  rq_init_comm_if_connected(9, "1")
  rq_init_comm_if_connected(2, "2")
  rq_init_comm_if_connected(3, "3")
  rq_init_comm_if_connected(4, "4")
  rq_print_connected_grippers()
  rq_gripper_communication_thread = run rq_gripper_communication()
  set_closed_norm(100.0, 1)
  set_open_norm(0.0, 1)
  set_closed_mm(0.0, 1)
  set_open_mm(50.0, 1)
  set_closed_norm(100.0, 2)
  set_open_norm(0.0, 2)
  set_closed_mm(0.0, 2)
  set_open_mm(50.0, 2)
  set_closed_norm(100.0, 3)
  set_open_norm(0.0, 3)
  set_closed_mm(0.0, 3)
  set_open_mm(50.0, 3)
  set_closed_norm(100.0, 4)
  set_open_norm(0.0, 4)
  set_closed_mm(0.0, 4)
  set_open_mm(50.0, 4)
  rq_current_limit_enabled = False
  while(not rq_gripper_communication_thread_started):
      sleep(0.008)
  end
  # end: URCap Installation Node
  step_count_6f5ccb1a_e640_4da3_bfd2_40e239d724c0 = 0.0
  thread Step_Counter_Thread_dce1a192_0697_4136_975c_3f443e1826c0():
    while (True):
      step_count_6f5ccb1a_e640_4da3_bfd2_40e239d724c0 = step_count_6f5ccb1a_e640_4da3_bfd2_40e239d724c0 + 1.0
      sync()
    end
  end
  run Step_Counter_Thread_dce1a192_0697_4136_975c_3f443e1826c0()
  global Pallet_1_cnt1=1
  global Pallet_1_lct=1
  global Pallet_1_lno=1
  global Pallet_1_sep= False
  global Pallet_1_tct=1
  global ready_bottle_01_p=p[.390695686427, .546143722526, .354784252936, -1.202154726952, -2.902476248553, -.000065055908]
  global ready_bottle_01_q=[1.2121562957763672, -1.5242460531047364, -1.8409428596496582, -1.3471840184978028, 1.569084882736206, -2.714905563985006]
  global Approach_p=p[.547491153120, .654222384983, -.068387800069, 1.202193147572, 2.902469227050, .000121933136]
  global Approach_q=[1.079941749572754, -2.4608241520323695, -1.818922519683838, -0.4325900834849854, 1.569946050643921, -2.84857422510256]
  global ToolActionPoint_p=p[.547456310296, .654165465094, -.466875056309, 1.202132749463, 2.902463524491, -.000036040777]
  global ToolActionPoint_q=[1.0798958534460201, -3.092485844440475, -1.4373697255328164, -0.182578185020553, 1.5701887189532613, -2.8485011726798497]
  global Exit_1_p=p[.547471692821, .654225285966, -.113240204994, 1.202149918204, 2.902456390812, .000132406260]
  global Exit_1_q=[1.0799791934124974, -2.5300233635810003, -1.7983936890644978, -0.38391026593322053, 1.5699977418301563, -2.8485885945959932]
  global other_side_botl_p=p[-.131302644250, .581179310947, .471637250643, 1.202107245272, 2.902505419242, .000006210820]
  global other_side_botl_q=[2.0894155502319336, -1.3711059850505372, -1.7675957679748535, -1.573710104028219, 1.5691683292388916, -1.8372095266925257]
  global bottle_insert_p=p[-.131260964550, .980471403249, .471604896898, 1.202196404184, 2.902428691936, .000004532766]
  global bottle_insert_q=[1.880312442779541, -2.055948873559469, -0.9804320335388184, -1.6760550938048304, 1.5698020458221436, -2.045520607625143]
  global bottle_placed_p=p[-.131258911804, .980469640209, .306164973509, -1.202200405733, -2.902392835778, -.000046866587]
  global bottle_placed_q=[1.880561113357544, -2.0672136745848597, -1.2540980577468872, -1.3910349768451233, 1.5695239305496216, -2.0459168593036097]
  global bottle_left_p=p[-.131220480029, .980475238550, .407942093095, -1.202222478666, -2.902455166129, -.000055421236]
  global bottle_left_q=[1.8803844451904297, -2.050185819665426, -1.1006345748901367, -1.5615647596171875, 1.5696470737457275, -2.0457008520709437]
  global Waypoint_1_p=p[-.642107095425, .666282486477, .300000000000, .017110052262, 3.141514691896, -.000101435305]
  global Waypoint_1_q=[2.5268598030394767, -1.9627318786897927, -1.4187371386550547, -1.331007934561983, 1.5694235174349547, -2.174366234433882]
  global towards_tool_p=p[-.319103721707, .922274672984, .289488424593, -2.161715004584, 2.087946977393, .189764243643]
  global towards_tool_q=[2.109555244445801, -2.0061499081053675, -1.4868388175964355, -1.0633927148631592, 1.4768521785736084, 2.067403554916382]
  global opener_release_p=p[-.319041217029, .960983395363, .063631881470, -2.151377132576, 2.078331762283, .208011082729]
  global opener_release_q=[2.0912246704101562, -2.235462804833883, -1.5705714225769043, -0.7327280801585694, 1.4711558818817139, 2.0473134517669678]
  global Waypoint_2_p=p[-.130580669380, .976983076115, .465670208769, -1.211351089344, 1.169811544850, 1.192461372640]
  global Waypoint_2_q=[2.048638343811035, -1.9488769970335902, -1.9945645332336426, 0.8238295751759033, 1.0946009159088135, -4.7583046595202845]
  global Waypoint_3_p=p[-.130500299950, .978149746807, .289697846114, -1.201141215498, 1.186848407184, 1.212169596068]
  global Waypoint_3_q=[2.046792984008789, -2.209787984887594, -2.0315918922424316, 1.1217116552540283, 1.098623514175415, -4.7331653277026575]
  global Waypoint_4_p=p[-.128825153461, .982323687907, .290256016280, -.673557451662, .725956132353, 1.488202477063]
  global Waypoint_4_q=[1.9992650747299194, -2.605262895623678, -1.638580322265625, 1.8312062460133056, 1.2280412912368774, -4.949915353451864]
  global Waypoint_7_p=p[-.128786997274, .992110967731, .291362608216, -.774623003114, .830703590919, 1.448526193777]
  global Waypoint_7_q=[2.0093674659729004, -2.5409466228880824, -1.719653606414795, 1.7121011453815917, 1.185677170753479, -4.909483496342794]
  global Waypoint_5_p=p[-.130885594544, .990636414244, .290303660438, -1.093247620272, 1.014798422788, 1.277726987509]
  global Waypoint_5_q=[2.0226666927337646, -2.338917394677633, -1.9369897842407227, 1.357553406352661, 1.154337763786316, -4.854938570653097]
  global Waypoint_6_p=p[-.129580234191, .994111291374, .289563055839, -1.211278069791, 1.169892183217, 1.192387357827]
  global Waypoint_6_q=[2.0349059104919434, -2.223354002038473, -1.9993042945861816, 1.1026395994373779, 1.1086199283599854, -4.757455412541525]
  global put_opener_back_p=p[-.319099897221, .974896383339, .066796819335, -2.237817946884, 2.161546728532, .045382917786]
  global put_opener_back_q=[2.062997817993164, -2.282285829583639, -1.4317312240600586, -0.9614525598338624, 1.549813985824585, 2.027625799179077]
  global release_opener_p=p[-.319054355550, .963210691229, .061049693193, -2.161547074700, 2.088102897465, .189944602177]
  global release_opener_q=[2.0875582695007324, -2.2436233959593714, -1.555147647857666, -0.7554741662791749, 1.4804890155792236, 2.045177698135376]
  $ 2 "BeforeStart"
  $ 3 "ready_to_take≔ False "
  global ready_to_take=  False
  $ 4 "Loop_1≔0"
  global Loop_1=0
  $ 5 "Set"
  set_tcp(p[0.0,0.0,0.195,0.0,0.0,0.0])
  thread EventThread():
    while (True):
      if (ready_to_take ==   True  ):
        $ 316 "Set Start=On"
        set_standard_digital_out(0, True)
        $ 317 "Wait: 0.25"
        sleep(0.25)
        $ 318 "Set Start=Off"
        set_standard_digital_out(0, False)
        $ 319 "Wait: 0.25"
        sleep(0.25)
        $ 320 "If bottle_sensor≟ False "
        if (get_standard_digital_in(1) ==   False  ):
          $ 321 "ready_to_take≔ False "
          global ready_to_take=  False
        end
      end
      sync()
    end
  end
  eventThread = run EventThread()
  $ 6 "Robot Program"
  # begin: URCap Program Node
  #   Source: triplea-wingman, 1.4.0, tripleA robotics ApS
  #   Type: AAA - Tools
  $ 7 "AAA - Tools"
  # end: URCap Program Node
  # begin: URCap Program Node
  #   Source: triplea-wingman, 1.4.0, tripleA robotics ApS
  #   Type: AAA - Get Tool
  $ 28 "AAA - Get T2           "
  $ 29 "Waypoints" "noBreak"
  $ 30 "tool_id_3≔'4a342d3e-ee93-4452-a102-fbcfc7771081'" "noBreak"
  global tool_id_3="4a342d3e-ee93-4452-a102-fbcfc7771081"
  $ 31 "tool_w1_3≔aaa_get_w(1, tool_id_3)" "noBreak"
  global tool_w1_3= aaa_get_w (1, tool_id_3)
  $ 32 "tool_w2_3≔aaa_get_w(2, tool_id_3)" "noBreak"
  global tool_w2_3= aaa_get_w (2, tool_id_3)
  $ 33 "tool_w3_3≔aaa_get_w(3, tool_id_3)" "noBreak"
  global tool_w3_3= aaa_get_w (3, tool_id_3)
  $ 34 "tool_w4_3≔aaa_get_w(4, tool_id_3)" "noBreak"
  global tool_w4_3= aaa_get_w (4, tool_id_3)
  $ 35 "tool_w0_3≔p[-0.6421144476781483, 0.6662879733766134, 0.20146973407971586, -0.017117761578530566, -3.1415327532565667, 1.0693642370029629E-4]" "noBreak"
  global tool_w0_3=p[-0.6421144476781483, 0.6662879733766134, 0.20146973407971586, -0.017117761578530566, -3.1415327532565667, 1.0693642370029629E-4]
  $ 36 "tool_w5_3≔p[-0.6421260084190709, 0.66626936215097, 0.20144070436964534, 0.01707995256586941, 3.1415293685776366, -1.3993269374544494E-4]" "noBreak"
  global tool_w5_3=p[-0.6421260084190709, 0.66626936215097, 0.20144070436964534, 0.01707995256586941, 3.1415293685776366, -1.3993269374544494E-4]
  $ 37 "Moving to Waypoints" "noBreak"
  $ 38 "'Setting Change TCP'" "noBreak"
  # 'Setting Change TCP'
  $ 39 "set_change_tc_3≔aaa_set_change_tcp(tool_id_3)" "noBreak"
  global set_change_tc_3= aaa_set_change_tcp (tool_id_3)
  $ 40 "'Setting Change Payload and Cog'" "noBreak"
  # 'Setting Change Payload and Cog'
  $ 41 "set_change_pc_3≔aaa_set_change_payload(tool_id_3)" "noBreak"
  global set_change_pc_3= aaa_set_change_payload (tool_id_3)
  $ 42 "'Enter Path'" "noBreak"
  # 'Enter Path'
  $ 43 "MoveL" "noBreak"
  $ 44 "tool_w0_3" "noBreak"
  movel(tool_w0_3, a=1.2, v=0.25)
  $ 45 "MoveL" "noBreak"
  $ 46 "tool_w1_3" "noBreak"
  movel(tool_w1_3, a=1.2, v=0.25)
  $ 47 "AAA script at W1" "noBreak"
  $ 48 "'Setting voltage to 0'" "noBreak"
  # 'Setting voltage to 0'
  $ 49 "set_w1_volt_3≔set_tool_voltage(0)" "noBreak"
  global set_w1_volt_3= set_tool_voltage (0)
  $ 50 "MoveL" "noBreak"
  $ 51 "tool_w2_3" "noBreak"
  movel(tool_w2_3, a=0.2, v=0.02)
  $ 52 "tool_w3_3" "noBreak"
  movel(tool_w3_3, a=0.2, v=0.02, r=0.01)
  $ 53 "Set User Payload and COG" "noBreak"
  $ 54 "set_user_pc_3≔aaa_set_user_payload(tool_id_3)" "noBreak"
  global set_user_pc_3= aaa_set_user_payload (tool_id_3)
  $ 55 "tool_w4_3" "noBreak"
  movel(tool_w4_3, a=0.2, v=0.02, r=0.005)
  $ 56 "AAA script at W4" "noBreak"
  $ 57 "'Using Standard Output'" "noBreak"
  # 'Using Standard Output'
  $ 58 "set_output_mo_1≔set_tool_output_mode(0)" "noBreak"
  global set_output_mo_1= set_tool_output_mode (0)
  $ 59 "set_dout_2≔set_tool_digital_output_mode(0, 2)" "noBreak"
  global set_dout_2= set_tool_digital_output_mode (0, 2)
  $ 60 "set_dout_3≔set_tool_digital_output_mode(1, 2)" "noBreak"
  global set_dout_3= set_tool_digital_output_mode (1, 2)
  $ 61 "set_tool_volt_3≔set_tool_voltage(24)" "noBreak"
  global set_tool_volt_3= set_tool_voltage (24)
  $ 62 "'Exit Path'" "noBreak"
  # 'Exit Path'
  $ 63 "MoveL" "noBreak"
  $ 64 "tool_w5_3" "noBreak"
  movel(tool_w5_3, a=1.2, v=0.25)
  $ 65 "Setting user TCP" "noBreak"
  $ 66 "set_user_tcp_1≔aaa_set_user_tcp(tool_id_3)" "noBreak"
  global set_user_tcp_1= aaa_set_user_tcp (tool_id_3)
  # end: URCap Program Node
  $ 67 "MoveJ"
  $ 68 "ready_bottle_01" "breakAfter"
  movej(get_inverse_kin(ready_bottle_01_p, qnear=ready_bottle_01_q), a=1.3962634015954636, v=1.0471975511965976)
  $ 69 "Loop 20 times"
  Loop_1 = 0
  while (Loop_1 < 20):
    $ 70 "Wait bottle_sensor=LO"
    while (get_standard_digital_in(1) == True):
      sync()
    end
    $ 71 "ready_to_take≔ False "
    global ready_to_take=  False
    $ 72 "Wait: 1.0"
    sleep(1.0)
    $ 73 "Set Start=On"
    set_standard_digital_out(0, True)
    $ 74 "Wait Start_buttom=HI"
    while (get_standard_digital_in(0) == False):
      sync()
    end
    $ 75 "Set Start=Off"
    set_standard_digital_out(0, False)
    $ 76 "Pallet_1"
    def Pallet_1_trans(pose):
    return p[pose[0], pose[1], pose[2], 0, 0, 0]
  end
  def Pallet_1_rot(pose):
  return p[0, 0, 0, pose[3], pose[4], pose[5]]
  end
  def Pallet_1_compute_pallet_waypoint(T_base_feature_taught, T_feature_referencePoint_taught, T_referencePoint_approach_taught, T_base_feature, T_base_referencePoint):
  local trans_referencePoint_approach_in_feature_taught = pose_sub(Pallet_1_trans(pose_trans(T_feature_referencePoint_taught, T_referencePoint_approach_taught)), Pallet_1_trans(T_feature_referencePoint_taught))
  local rot_referencePoint_approach_in_feature_taught = pose_trans(Pallet_1_rot(T_feature_referencePoint_taught), pose_trans(Pallet_1_rot(T_referencePoint_approach_taught), pose_inv(Pallet_1_rot(T_feature_referencePoint_taught))))
  T_feature_referencePoint = pose_trans(pose_inv(T_base_feature), T_base_referencePoint)
  rot_referencePoint_approach = pose_trans(pose_inv(Pallet_1_rot(T_feature_referencePoint)), pose_trans(rot_referencePoint_approach_in_feature_taught, Pallet_1_rot(T_feature_referencePoint)))
  T_feature_approach = pose_trans(trans_referencePoint_approach_in_feature_taught, pose_trans(T_feature_referencePoint, rot_referencePoint_approach))
  T_base_approach = pose_trans(T_base_feature, T_feature_approach)
  return T_base_approach
  end
  Pallet_1_tct = 20
  if (Pallet_1_cnt1 > 20 or Pallet_1_cnt1 < 1):
    Pallet_1_cnt1 = 1
  end
  $ 77 "Patterns" "noBreak"
  $ 78 "Bierkisten" "noBreak"
  $ 83 "Layers" "noBreak"
  if (Pallet_1_cnt1 < 21):
    Pallet_1_lno = 1
    Pallet_1_lct = Pallet_1_cnt1
    global CornerItem_1=pose_trans(p[0.0,0.0,0.0,0.0,0.0,0.0], pose_trans(p[-.000000000000, -.000000000000, -.000000000000, .000000000000, .000000000000, .000000000000], p[.547456310296, .654165465094, -.466875056309, 1.202132749464, 2.902463524495, -.000036040781]))
    global CornerItem_2=pose_trans(p[0.0,0.0,0.0,0.0,0.0,0.0], pose_trans(p[-.000000000000, -.000000000000, -.000000000000, .000000000000, .000000000000, .000000000000], p[.255583455772, .658553152541, -.466885764013, 1.202183125409, 2.902424122183, .000039330012]))
    global CornerItem_3=pose_trans(p[0.0,0.0,0.0,0.0,0.0,0.0], pose_trans(p[-.000000000000, -.000000000000, -.000000000000, .000000000000, .000000000000, .000000000000], p[.252284532779, .448281458720, -.466787023823, -1.198647047037, -2.893601694178, .004266709226]))
    global CornerItem_4=pose_trans(p[0.0,0.0,0.0,0.0,0.0,0.0], pose_trans(p[-.000000000000, -.000000000000, -.000000000000, .000000000000, .000000000000, .000000000000], p[.547223255359, .446272651206, -.466853397510, -1.202135566826, -2.902466008849, -.000024200332]))
    Pallet_1_cnt1_x = (Pallet_1_lct - 1) % 5
    Pallet_1_cnt1_y = floor((Pallet_1_lct - 1) / 5)
    referencePoint = interpolate_pose(interpolate_pose(CornerItem_1, CornerItem_2, Pallet_1_cnt1_x/4), interpolate_pose(CornerItem_4, CornerItem_3,Pallet_1_cnt1_x/4), Pallet_1_cnt1_y/3)
    direction = p[0,0,1,0,0,0]
    referencePoint = pose_add (referencePoint,p[0.0*direction[0],0.0*direction[1],0.0*direction[2],0,0,0])
  end
  Approach_p = Pallet_1_compute_pallet_waypoint(p[0.0,0.0,0.0,0.0,0.0,0.0], pose_trans(pose_inv(p[0.0,0.0,0.0,0.0,0.0,0.0]), p[0.5474563102958362,0.6541654650937244,-0.46687505630886694,1.202132749464188,2.90246352449483,-3.604078102808996E-5]), p[1.1660793748785592E-6,6.097173717700688E-5,-0.3984872571625544,-8.205397251571686E-5,6.470613541237836E-5,3.4136223316427125E-5], p[0.0,0.0,0.0,0.0,0.0,0.0], referencePoint)
  Approach_p = pose_trans(p[0.5474563102958362,0.6541654650937244,-0.46687505630886694,1.2021327494670466,2.902463524501732,-3.6040774637205476E-5], pose_trans(pose_inv(referencePoint), Approach_p))
  ToolActionPoint_p = Pallet_1_compute_pallet_waypoint(p[0.0,0.0,0.0,0.0,0.0,0.0], pose_trans(pose_inv(p[0.0,0.0,0.0,0.0,0.0,0.0]), p[0.5474563102958362,0.6541654650937244,-0.46687505630886694,1.202132749464188,2.90246352449483,-3.604078102808996E-5]), p[-5.551115123125783E-17,-1.1102230246251565E-16,0.0,-2.7441461671829574E-12,-1.099368366185168E-11,3.5712370008347063E-13], p[0.0,0.0,0.0,0.0,0.0,0.0], referencePoint)
  ToolActionPoint_p = pose_trans(p[0.5474563102958362,0.6541654650937244,-0.46687505630886694,1.2021327494670466,2.902463524501732,-3.6040774637205476E-5], pose_trans(pose_inv(referencePoint), ToolActionPoint_p))
  Exit_1_p = Pallet_1_compute_pallet_waypoint(p[0.0,0.0,0.0,0.0,0.0,0.0], pose_trans(pose_inv(p[0.0,0.0,0.0,0.0,0.0,0.0]), p[0.5474563102958362,0.6541654650937244,-0.46687505630886694,1.202132749464188,2.90246352449483,-3.604078102808996E-5]), p[1.860402541670192E-5,4.970421858563334E-5,-0.3536348527263402,-9.908286752325829E-5,4.1018018506442885E-5,1.1837606331770305E-5], p[0.0,0.0,0.0,0.0,0.0,0.0], referencePoint)
  Exit_1_p = pose_trans(p[0.5474563102958362,0.6541654650937244,-0.46687505630886694,1.2021327494670466,2.902463524501732,-3.6040774637205476E-5], pose_trans(pose_inv(referencePoint), Exit_1_p))
  $ 84 "At Each Item" "noBreak"
  $ 85 "Generated Movements" "noBreak"
  $ 86 "MoveJ" "noBreak"
  $ 87 "Approach" "noBreak"
  movej(get_inverse_kin(pose_trans(referencePoint, pose_trans(p[-.075418209057, -.849684240225, -.466863975119, -1.202132749467, -2.902463524502, .000036040775], Approach_p)), qnear=Approach_q), a=1.3962634015954636, v=1.0471975511965976)
  $ 88 "MoveL" "noBreak"
  $ 89 "ToolActionPoint" "noBreak"
  movel(pose_trans(referencePoint, pose_trans(p[-.075418209057, -.849684240225, -.466863975119, -1.202132749467, -2.902463524502, .000036040775], ToolActionPoint_p)), a=1.2, v=0.15)
  $ 90 "Tool action" "noBreak"
  $ 91 "Set TO[1]=Off" "noBreak"
  set_tool_digital_out(1, False)
  $ 92 "Wait: 0.15" "noBreak"
  sleep(0.15)
  $ 93 "Set TO[0]=On" "noBreak"
  set_tool_digital_out(0, True)
  $ 94 "Wait: 1.0" "noBreak"
  sleep(1.0)
  $ 95 "MoveL" "noBreak"
  $ 96 "Exit_1" "noBreak"
  movel(pose_trans(referencePoint, pose_trans(p[-.075418209057, -.849684240225, -.466863975119, -1.202132749467, -2.902463524502, .000036040775], Exit_1_p)), a=1.2, v=0.25)
  Pallet_1_sep = False
  if (Pallet_1_cnt1 >= 20):
    Pallet_1_cnt1 = 1
  else:
    Pallet_1_cnt1 = Pallet_1_cnt1 + 1
  end
  $ 97 "MoveL"
  $ 98 "ready_bottle_01" "breakAfter"
  movel(ready_bottle_01_p, a=1.0, v=0.3)
  $ 99 "other_side_botl" "breakAfter"
  movel(other_side_botl_p, a=1.0, v=0.3)
  $ 100 "bottle_insert" "breakAfter"
  movel(bottle_insert_p, a=1.0, v=0.3)
  $ 101 "bottle_placed" "breakAfter"
  movel(bottle_placed_p, a=1.2, v=0.05)
  $ 102 "Set TO[0]=Off"
  set_tool_digital_out(0, False)
  $ 103 "Wait: 0.15"
  sleep(0.15)
  $ 104 "Set TO[1]=On"
  set_tool_digital_out(1, True)
  $ 105 "Wait: 0.5"
  sleep(0.5)
  $ 106 "bottle_left" "breakAfter"
  movel(bottle_left_p, a=1.0, v=0.3)
  # begin: URCap Program Node
  #   Source: triplea-wingman, 1.4.0, tripleA robotics ApS
  #   Type: AAA - Put Tool
  $ 107 "AAA - Put T2           "
  $ 108 "Waypoints" "noBreak"
  $ 109 "tool_id_4≔'4a342d3e-ee93-4452-a102-fbcfc7771081'" "noBreak"
  global tool_id_4="4a342d3e-ee93-4452-a102-fbcfc7771081"
  $ 110 "tool_w1_4≔aaa_get_w(1, tool_id_4)" "noBreak"
  global tool_w1_4= aaa_get_w (1, tool_id_4)
  $ 111 "tool_w2_4≔aaa_get_w(2, tool_id_4)" "noBreak"
  global tool_w2_4= aaa_get_w (2, tool_id_4)
  $ 112 "tool_w3_4≔aaa_get_w(3, tool_id_4)" "noBreak"
  global tool_w3_4= aaa_get_w (3, tool_id_4)
  $ 113 "tool_w4_4≔aaa_get_w(4, tool_id_4)" "noBreak"
  global tool_w4_4= aaa_get_w (4, tool_id_4)
  $ 114 "tool_w0_4≔p[-0.6421144476781483, 0.6662879733766134, 0.20146973407971586, -0.017117761578530566, -3.1415327532565667, 1.0693642370029629E-4]" "noBreak"
  global tool_w0_4=p[-0.6421144476781483, 0.6662879733766134, 0.20146973407971586, -0.017117761578530566, -3.1415327532565667, 1.0693642370029629E-4]
  $ 115 "tool_w5_4≔p[-0.6421260084190709, 0.66626936215097, 0.20144070436964534, 0.01707995256586941, 3.1415293685776366, -1.3993269374544494E-4]" "noBreak"
  global tool_w5_4=p[-0.6421260084190709, 0.66626936215097, 0.20144070436964534, 0.01707995256586941, 3.1415293685776366, -1.3993269374544494E-4]
  $ 116 "Moving to Waypoints" "noBreak"
  $ 117 "'Setting Change TCP'" "noBreak"
  # 'Setting Change TCP'
  $ 118 "set_change_tc_4≔aaa_set_change_tcp(tool_id_4)" "noBreak"
  global set_change_tc_4= aaa_set_change_tcp (tool_id_4)
  $ 119 "set_user_pc_4≔aaa_set_user_payload(tool_id_4)" "noBreak"
  global set_user_pc_4= aaa_set_user_payload (tool_id_4)
  $ 120 "'Exit Path'" "noBreak"
  # 'Exit Path'
  $ 121 "MoveL" "noBreak"
  $ 122 "tool_w5_4" "noBreak"
  movel(tool_w5_4, a=1.2, v=0.25)
  $ 123 "MoveL" "noBreak"
  $ 124 "tool_w4_4" "noBreak"
  movel(tool_w4_4, a=1.2, v=0.25, r=0.005)
  $ 125 "AAA script at W4" "noBreak"
  $ 126 "set_tool_volt_4≔set_tool_voltage(0)" "noBreak"
  global set_tool_volt_4= set_tool_voltage (0)
  $ 127 "MoveL" "noBreak"
  $ 128 "tool_w3_4" "noBreak"
  movel(tool_w3_4, a=0.2, v=0.02, r=0.01)
  $ 129 "Set Change Payload and COG" "noBreak"
  $ 130 "set_change_pc_4≔aaa_set_change_payload(tool_id_4)" "noBreak"
  global set_change_pc_4= aaa_set_change_payload (tool_id_4)
  $ 131 "tool_w2_4" "noBreak"
  movel(tool_w2_4, a=0.2, v=0.02)
  $ 132 "AAA script at W1" "noBreak"
  $ 133 "'Setting voltage to 0'" "noBreak"
  # 'Setting voltage to 0'
  $ 134 "set_w1_volt_4≔set_tool_voltage(0)" "noBreak"
  global set_w1_volt_4= set_tool_voltage (0)
  $ 135 "tool_w1_4" "noBreak"
  movel(tool_w1_4, a=0.2, v=0.02)
  $ 136 "'Enter Path'" "noBreak"
  # 'Enter Path'
  $ 137 "MoveL" "noBreak"
  $ 138 "tool_w0_4" "noBreak"
  movel(tool_w0_4, a=1.2, v=0.25)
  # end: URCap Program Node
  # begin: URCap Program Node
  #   Source: triplea-wingman, 1.4.0, tripleA robotics ApS
  #   Type: AAA - Get Tool
  $ 139 "AAA - Get Robotiq_e           "
  $ 140 "Waypoints" "noBreak"
  $ 141 "tool_id≔'4b514240-cf4e-4bf1-8bd0-419c27a4d488'" "noBreak"
  global tool_id="4b514240-cf4e-4bf1-8bd0-419c27a4d488"
  $ 142 "tool_w1≔aaa_get_w(1, tool_id)" "noBreak"
  global tool_w1= aaa_get_w (1, tool_id)
  $ 143 "tool_w2≔aaa_get_w(2, tool_id)" "noBreak"
  global tool_w2= aaa_get_w (2, tool_id)
  $ 144 "tool_w3≔aaa_get_w(3, tool_id)" "noBreak"
  global tool_w3= aaa_get_w (3, tool_id)
  $ 145 "tool_w4≔aaa_get_w(4, tool_id)" "noBreak"
  global tool_w4= aaa_get_w (4, tool_id)
  $ 146 "tool_w0≔p[-0.6421231560845492, 0.6662690344927905, 0.20142700950352788, 0.017023535316556416, 3.141493526432438, -1.5673970200807575E-4]" "noBreak"
  global tool_w0=p[-0.6421231560845492, 0.6662690344927905, 0.20142700950352788, 0.017023535316556416, 3.141493526432438, -1.5673970200807575E-4]
  $ 147 "tool_w5≔p[-0.6421151581475879, 0.6662702288012549, 0.20146681548744672, -0.01704285243180614, -3.1415231156302963, 1.6352643870166494E-4]" "noBreak"
  global tool_w5=p[-0.6421151581475879, 0.6662702288012549, 0.20146681548744672, -0.01704285243180614, -3.1415231156302963, 1.6352643870166494E-4]
  $ 148 "Moving to Waypoints" "noBreak"
  $ 149 "'Setting Change TCP'" "noBreak"
  # 'Setting Change TCP'
  $ 150 "set_change_tcp≔aaa_set_change_tcp(tool_id)" "noBreak"
  global set_change_tcp= aaa_set_change_tcp (tool_id)
  $ 151 "'Setting Change Payload and Cog'" "noBreak"
  # 'Setting Change Payload and Cog'
  $ 152 "set_change_pc≔aaa_set_change_payload(tool_id)" "noBreak"
  global set_change_pc= aaa_set_change_payload (tool_id)
  $ 153 "'Enter Path'" "noBreak"
  # 'Enter Path'
  $ 154 "MoveL" "noBreak"
  $ 155 "tool_w0" "noBreak"
  movel(tool_w0, a=1.2, v=0.25)
  $ 156 "MoveL" "noBreak"
  $ 157 "tool_w1" "noBreak"
  movel(tool_w1, a=1.2, v=0.25)
  $ 158 "AAA script at W1" "noBreak"
  $ 159 "'Setting voltage to 0'" "noBreak"
  # 'Setting voltage to 0'
  $ 160 "set_w1_volt≔set_tool_voltage(0)" "noBreak"
  global set_w1_volt= set_tool_voltage (0)
  $ 161 "MoveL" "noBreak"
  $ 162 "tool_w2" "noBreak"
  movel(tool_w2, a=0.2, v=0.02)
  $ 163 "tool_w3" "noBreak"
  movel(tool_w3, a=0.2, v=0.02, r=0.01)
  $ 164 "Set User Payload and COG" "noBreak"
  $ 165 "set_user_pc≔aaa_set_user_payload(tool_id)" "noBreak"
  global set_user_pc= aaa_set_user_payload (tool_id)
  $ 166 "tool_w4" "noBreak"
  movel(tool_w4, a=0.2, v=0.02, r=0.005)
  $ 167 "AAA script at W4" "noBreak"
  $ 168 "'Using Standard Output'" "noBreak"
  # 'Using Standard Output'
  $ 169 "set_output_mode≔set_tool_output_mode(0)" "noBreak"
  global set_output_mode= set_tool_output_mode (0)
  $ 170 "set_dout_0≔set_tool_digital_output_mode(0, 1)" "noBreak"
  global set_dout_0= set_tool_digital_output_mode (0, 1)
  $ 171 "set_dout_1≔set_tool_digital_output_mode(1, 1)" "noBreak"
  global set_dout_1= set_tool_digital_output_mode (1, 1)
  $ 172 "set_tool_volt≔set_tool_voltage(24)" "noBreak"
  global set_tool_volt= set_tool_voltage (24)
  $ 173 "'Exit Path'" "noBreak"
  # 'Exit Path'
  $ 174 "MoveL" "noBreak"
  $ 175 "tool_w5" "noBreak"
  movel(tool_w5, a=1.2, v=0.25)
  $ 176 "Setting user TCP" "noBreak"
  $ 177 "set_user_tcp≔aaa_set_user_tcp(tool_id)" "noBreak"
  global set_user_tcp= aaa_set_user_tcp (tool_id)
  $ 178 "Wait: 4.0" "noBreak"
  sleep(4.0)
  # begin: URCap Program Node
  #   Source: Robotiq_Grippers, 1.8.13.22852, Robotiq Inc.
  #   Type: Gripper Activate
  $ 179 "Gripper Activate" "noBreak"

  kill rq_gripper_communication_thread
  rq_gripper_communication_thread_started = False
  rq_close_gripper_socket("1")
  rq_close_gripper_socket("2")
  rq_close_gripper_socket("3")
  rq_close_gripper_socket("4")

  rq_init_comm_if_connected(9, "1")
  rq_init_comm_if_connected(2, "2")
  rq_init_comm_if_connected(3, "3")
  rq_init_comm_if_connected(4, "4")
  rq_print_connected_grippers()
  rq_gripper_communication_thread = run rq_gripper_communication()

  while(not rq_gripper_communication_thread_started):
      sleep(0.008)
  end

  rq_set_max_current_for_all_grippers()

  reset_and_activate = False

  rq_activate_all_grippers(False)
  # end: URCap Program Node
  $ 180 "If rq_is_gripper_connected()≟ False " "noBreak"
  if (rq_is_gripper_connected() ==   False  ):
    $ 181 "Wait: 2.0" "noBreak"
    sleep(2.0)
    # begin: URCap Program Node
    #   Source: Robotiq_Grippers, 1.8.13.22852, Robotiq Inc.
    #   Type: Gripper Activate
    $ 182 "Gripper Reset and Activate" "noBreak"

    kill rq_gripper_communication_thread
    rq_gripper_communication_thread_started = False
    rq_close_gripper_socket("1")
    rq_close_gripper_socket("2")
    rq_close_gripper_socket("3")
    rq_close_gripper_socket("4")

    rq_init_comm_if_connected(9, "1")
    rq_init_comm_if_connected(2, "2")
    rq_init_comm_if_connected(3, "3")
    rq_init_comm_if_connected(4, "4")
    rq_print_connected_grippers()
    rq_gripper_communication_thread = run rq_gripper_communication()

    while(not rq_gripper_communication_thread_started):
        sleep(0.008)
    end

    rq_set_max_current_for_all_grippers()

    reset_and_activate = True

    rq_activate_all_grippers(True)
    # end: URCap Program Node
  end
  # end: URCap Program Node
  $ 183 "MoveL"
  $ 184 "Waypoint_1" "breakAfter"
  movel(Waypoint_1_p, a=1.0, v=0.3)
  $ 185 "towards_tool" "breakAfter"
  movel(towards_tool_p, a=1.0, v=0.3)
  $ 186 "Set"
  set_tcp(p[0.0,0.0,0.157,0.0,0.0,0.0])
  $ 187 "opener_release" "breakAfter"
  movel(opener_release_p, a=1.0, v=0.3)
  # begin: URCap Program Node
  #   Source: Robotiq_Grippers, 1.8.13.22852, Robotiq Inc.
  #   Type: Gripper
  $ 188 "Gripper Close (1)"
  if not(gripper_connected[0]):
    popup("Gripper 1 must be connected to run this program.", "No connection", False, True, True)
  end
  if not(rq_is_gripper_activated("1")):
    popup("Gripper 1 is not activated. Go to Installation tab > Gripper to activate it and run the program again.", "Not activated", False, True, True)
  end
  rq_set_pos_spd_for(255, 255, 255, "1")
  rq_wait_pos_spe_for_request(255, 255, 255, "1")
  rq_go_to("1")
  rq_wait("1")
  # end: URCap Program Node
  $ 189 "towards_tool" "breakAfter"
  movel(towards_tool_p, a=1.0, v=0.3)
  $ 190 "Set"
  set_tcp(p[0.0,0.0,0.23,0.0,0.0,0.0])
  $ 191 "Set Payload: 5.000kg CoG=[0.00mm, 0.00mm, 0.00mm]"
  set_target_payload(5.000000, [0.000000, 0.000000, 0.000000], [0.022505, 0.022505, 0.022505, 0.000000, 0.000000, 0.000000])
  $ 192 "Waypoint_2" "breakAfter"
  movel(Waypoint_2_p, a=1.0, v=0.3)
  $ 193 "Waypoint_3" "breakAfter"
  movel(Waypoint_3_p, a=1.0, v=0.3)
  $ 194 "Waypoint_4" "breakAfter"
  movel(Waypoint_4_p, a=1.0, v=0.05)
  $ 195 "Waypoint_7" "breakAfter"
  movel(Waypoint_7_p, a=1.0, v=0.05)
  $ 196 "Waypoint_5" "breakAfter"
  movel(Waypoint_5_p, a=1.0, v=0.05)
  $ 197 "Waypoint_6" "breakAfter"
  movel(Waypoint_6_p, a=1.0, v=0.05)
  $ 198 "Waypoint_2" "breakAfter"
  movel(Waypoint_2_p, a=1.0, v=0.3)
  $ 199 "towards_tool" "breakAfter"
  movel(towards_tool_p, a=1.0, v=0.3)
  $ 200 "Set"
  set_tcp(p[0.0,0.0,0.157,0.0,0.0,0.0])
  $ 201 "Set Payload: Payload"
  set_target_payload(0.150000, [0.000000, 0.000000, 0.100000], [0.000000, 0.000000, 0.000000, 0.000000, 0.000000, 0.000000])
  $ 202 "put_opener_back" "breakAfter"
  movel(put_opener_back_p, a=1.0, v=0.3)
  $ 203 "ready_to_take≔ True "
  global ready_to_take=  True
  $ 204 "opener_release" "breakAfter"
  movel(opener_release_p, a=1.0, v=0.3)
  # begin: URCap Program Node
  #   Source: Robotiq_Grippers, 1.8.13.22852, Robotiq Inc.
  #   Type: Gripper
  $ 205 "Gripper Move50% (1)"
  if not(gripper_connected[0]):
    popup("Gripper 1 must be connected to run this program.", "No connection", False, True, True)
  end
  if not(rq_is_gripper_activated("1")):
    popup("Gripper 1 is not activated. Go to Installation tab > Gripper to activate it and run the program again.", "Not activated", False, True, True)
  end
  rq_set_pos_spd_for(128, 0, 0, "1")
  rq_wait_pos_spe_for_request(128, 0, 0, "1")
  rq_go_to("1")
  rq_wait("1")
  # end: URCap Program Node
  $ 206 "release_opener" "breakAfter"
  movel(release_opener_p, a=1.0, v=0.3)
  # begin: URCap Program Node
  #   Source: Robotiq_Grippers, 1.8.13.22852, Robotiq Inc.
  #   Type: Gripper
  $ 207 "Gripper Open (1)"
  if not(gripper_connected[0]):
    popup("Gripper 1 must be connected to run this program.", "No connection", False, True, True)
  end
  if not(rq_is_gripper_activated("1")):
    popup("Gripper 1 is not activated. Go to Installation tab > Gripper to activate it and run the program again.", "Not activated", False, True, True)
  end
  rq_set_pos_spd_for(0, 255, 255, "1")
  rq_wait_pos_spe_for_request(0, 255, 255, "1")
  rq_go_to("1")
  rq_wait("1")
  # end: URCap Program Node
  $ 208 "towards_tool" "breakAfter"
  movel(towards_tool_p, a=1.0, v=0.3)
  $ 209 "Waypoint_1" "breakAfter"
  movel(Waypoint_1_p, a=1.0, v=0.3)
  # begin: URCap Program Node
  #   Source: triplea-wingman, 1.4.0, tripleA robotics ApS
  #   Type: AAA - Put Tool
  $ 210 "AAA - Put Robotiq_e           "
  $ 211 "Waypoints" "noBreak"
  $ 212 "tool_id_7≔'4b514240-cf4e-4bf1-8bd0-419c27a4d488'" "noBreak"
  global tool_id_7="4b514240-cf4e-4bf1-8bd0-419c27a4d488"
  $ 213 "tool_w1_7≔aaa_get_w(1, tool_id_7)" "noBreak"
  global tool_w1_7= aaa_get_w (1, tool_id_7)
  $ 214 "tool_w2_7≔aaa_get_w(2, tool_id_7)" "noBreak"
  global tool_w2_7= aaa_get_w (2, tool_id_7)
  $ 215 "tool_w3_7≔aaa_get_w(3, tool_id_7)" "noBreak"
  global tool_w3_7= aaa_get_w (3, tool_id_7)
  $ 216 "tool_w4_7≔aaa_get_w(4, tool_id_7)" "noBreak"
  global tool_w4_7= aaa_get_w (4, tool_id_7)
  $ 217 "tool_w0_7≔p[-0.6421231560845492, 0.6662690344927905, 0.20142700950352788, 0.017023535316556416, 3.141493526432438, -1.5673970200807575E-4]" "noBreak"
  global tool_w0_7=p[-0.6421231560845492, 0.6662690344927905, 0.20142700950352788, 0.017023535316556416, 3.141493526432438, -1.5673970200807575E-4]
  $ 218 "tool_w5_7≔p[-0.6421151581475879, 0.6662702288012549, 0.20146681548744672, -0.01704285243180614, -3.1415231156302963, 1.6352643870166494E-4]" "noBreak"
  global tool_w5_7=p[-0.6421151581475879, 0.6662702288012549, 0.20146681548744672, -0.01704285243180614, -3.1415231156302963, 1.6352643870166494E-4]
  $ 219 "Moving to Waypoints" "noBreak"
  $ 220 "'Setting Change TCP'" "noBreak"
  # 'Setting Change TCP'
  $ 221 "set_change_tc_7≔aaa_set_change_tcp(tool_id_7)" "noBreak"
  global set_change_tc_7= aaa_set_change_tcp (tool_id_7)
  $ 222 "set_user_pc_7≔aaa_set_user_payload(tool_id_7)" "noBreak"
  global set_user_pc_7= aaa_set_user_payload (tool_id_7)
  $ 223 "'Exit Path'" "noBreak"
  # 'Exit Path'
  $ 224 "MoveL" "noBreak"
  $ 225 "tool_w5_7" "noBreak"
  movel(tool_w5_7, a=1.2, v=0.25)
  $ 226 "MoveL" "noBreak"
  $ 227 "tool_w4_7" "noBreak"
  movel(tool_w4_7, a=1.2, v=0.25, r=0.005)
  $ 228 "AAA script at W4" "noBreak"
  $ 229 "set_tool_volt_7≔set_tool_voltage(0)" "noBreak"
  global set_tool_volt_7= set_tool_voltage (0)
  $ 230 "MoveL" "noBreak"
  $ 231 "tool_w3_7" "noBreak"
  movel(tool_w3_7, a=0.2, v=0.02, r=0.01)
  $ 232 "Set Change Payload and COG" "noBreak"
  $ 233 "set_change_pc_7≔aaa_set_change_payload(tool_id_7)" "noBreak"
  global set_change_pc_7= aaa_set_change_payload (tool_id_7)
  $ 234 "tool_w2_7" "noBreak"
  movel(tool_w2_7, a=0.2, v=0.02)
  $ 235 "AAA script at W1" "noBreak"
  $ 236 "'Setting voltage to 0'" "noBreak"
  # 'Setting voltage to 0'
  $ 237 "set_w1_volt_7≔set_tool_voltage(0)" "noBreak"
  global set_w1_volt_7= set_tool_voltage (0)
  $ 238 "tool_w1_7" "noBreak"
  movel(tool_w1_7, a=0.2, v=0.02)
  $ 239 "'Enter Path'" "noBreak"
  # 'Enter Path'
  $ 240 "MoveL" "noBreak"
  $ 241 "tool_w0_7" "noBreak"
  movel(tool_w0_7, a=1.2, v=0.25)
  # end: URCap Program Node
  # begin: URCap Program Node
  #   Source: triplea-wingman, 1.4.0, tripleA robotics ApS
  #   Type: AAA - Get Tool
  $ 242 "AAA - Get T2           "
  $ 243 "Waypoints" "noBreak"
  $ 244 "tool_id_5≔'4a342d3e-ee93-4452-a102-fbcfc7771081'" "noBreak"
  global tool_id_5="4a342d3e-ee93-4452-a102-fbcfc7771081"
  $ 245 "tool_w1_5≔aaa_get_w(1, tool_id_5)" "noBreak"
  global tool_w1_5= aaa_get_w (1, tool_id_5)
  $ 246 "tool_w2_5≔aaa_get_w(2, tool_id_5)" "noBreak"
  global tool_w2_5= aaa_get_w (2, tool_id_5)
  $ 247 "tool_w3_5≔aaa_get_w(3, tool_id_5)" "noBreak"
  global tool_w3_5= aaa_get_w (3, tool_id_5)
  $ 248 "tool_w4_5≔aaa_get_w(4, tool_id_5)" "noBreak"
  global tool_w4_5= aaa_get_w (4, tool_id_5)
  $ 249 "tool_w0_5≔p[-0.6421144476781483, 0.6662879733766134, 0.20146973407971586, -0.017117761578530566, -3.1415327532565667, 1.0693642370029629E-4]" "noBreak"
  global tool_w0_5=p[-0.6421144476781483, 0.6662879733766134, 0.20146973407971586, -0.017117761578530566, -3.1415327532565667, 1.0693642370029629E-4]
  $ 250 "tool_w5_5≔p[-0.6421260084190709, 0.66626936215097, 0.20144070436964534, 0.01707995256586941, 3.1415293685776366, -1.3993269374544494E-4]" "noBreak"
  global tool_w5_5=p[-0.6421260084190709, 0.66626936215097, 0.20144070436964534, 0.01707995256586941, 3.1415293685776366, -1.3993269374544494E-4]
  $ 251 "Moving to Waypoints" "noBreak"
  $ 252 "'Setting Change TCP'" "noBreak"
  # 'Setting Change TCP'
  $ 253 "set_change_tc_5≔aaa_set_change_tcp(tool_id_5)" "noBreak"
  global set_change_tc_5= aaa_set_change_tcp (tool_id_5)
  $ 254 "'Setting Change Payload and Cog'" "noBreak"
  # 'Setting Change Payload and Cog'
  $ 255 "set_change_pc_5≔aaa_set_change_payload(tool_id_5)" "noBreak"
  global set_change_pc_5= aaa_set_change_payload (tool_id_5)
  $ 256 "'Enter Path'" "noBreak"
  # 'Enter Path'
  $ 257 "MoveL" "noBreak"
  $ 258 "tool_w0_5" "noBreak"
  movel(tool_w0_5, a=1.2, v=0.25)
  $ 259 "MoveL" "noBreak"
  $ 260 "tool_w1_5" "noBreak"
  movel(tool_w1_5, a=1.2, v=0.25)
  $ 261 "AAA script at W1" "noBreak"
  $ 262 "'Setting voltage to 0'" "noBreak"
  # 'Setting voltage to 0'
  $ 263 "set_w1_volt_5≔set_tool_voltage(0)" "noBreak"
  global set_w1_volt_5= set_tool_voltage (0)
  $ 264 "MoveL" "noBreak"
  $ 265 "tool_w2_5" "noBreak"
  movel(tool_w2_5, a=0.2, v=0.02)
  $ 266 "tool_w3_5" "noBreak"
  movel(tool_w3_5, a=0.2, v=0.02, r=0.01)
  $ 267 "Set User Payload and COG" "noBreak"
  $ 268 "set_user_pc_5≔aaa_set_user_payload(tool_id_5)" "noBreak"
  global set_user_pc_5= aaa_set_user_payload (tool_id_5)
  $ 269 "tool_w4_5" "noBreak"
  movel(tool_w4_5, a=0.2, v=0.02, r=0.005)
  $ 270 "AAA script at W4" "noBreak"
  $ 271 "'Using Standard Output'" "noBreak"
  # 'Using Standard Output'
  $ 272 "set_output_mo_4≔set_tool_output_mode(0)" "noBreak"
  global set_output_mo_4= set_tool_output_mode (0)
  $ 273 "set_dout_8≔set_tool_digital_output_mode(0, 2)" "noBreak"
  global set_dout_8= set_tool_digital_output_mode (0, 2)
  $ 274 "set_dout_9≔set_tool_digital_output_mode(1, 2)" "noBreak"
  global set_dout_9= set_tool_digital_output_mode (1, 2)
  $ 275 "set_tool_volt_5≔set_tool_voltage(24)" "noBreak"
  global set_tool_volt_5= set_tool_voltage (24)
  $ 276 "'Exit Path'" "noBreak"
  # 'Exit Path'
  $ 277 "MoveL" "noBreak"
  $ 278 "tool_w5_5" "noBreak"
  movel(tool_w5_5, a=1.2, v=0.25)
  $ 279 "Setting user TCP" "noBreak"
  $ 280 "set_user_tcp_4≔aaa_set_user_tcp(tool_id_5)" "noBreak"
  global set_user_tcp_4= aaa_set_user_tcp (tool_id_5)
  # end: URCap Program Node
  $ 281 "other_side_botl" "breakAfter"
  movel(other_side_botl_p, a=1.0, v=0.3)
  $ 282 "ready_bottle_01" "breakAfter"
  movel(ready_bottle_01_p, a=1.0, v=0.3)
  Loop_1 = Loop_1 + 1
  end
  # begin: URCap Program Node
  #   Source: triplea-wingman, 1.4.0, tripleA robotics ApS
  #   Type: AAA - Put Tool
  $ 283 "AAA - Put T2           "
  $ 284 "Waypoints" "noBreak"
  $ 285 "tool_id_6≔'4a342d3e-ee93-4452-a102-fbcfc7771081'" "noBreak"
  global tool_id_6="4a342d3e-ee93-4452-a102-fbcfc7771081"
  $ 286 "tool_w1_6≔aaa_get_w(1, tool_id_6)" "noBreak"
  global tool_w1_6= aaa_get_w (1, tool_id_6)
  $ 287 "tool_w2_6≔aaa_get_w(2, tool_id_6)" "noBreak"
  global tool_w2_6= aaa_get_w (2, tool_id_6)
  $ 288 "tool_w3_6≔aaa_get_w(3, tool_id_6)" "noBreak"
  global tool_w3_6= aaa_get_w (3, tool_id_6)
  $ 289 "tool_w4_6≔aaa_get_w(4, tool_id_6)" "noBreak"
  global tool_w4_6= aaa_get_w (4, tool_id_6)
  $ 290 "tool_w0_6≔p[-0.6421144476781483, 0.6662879733766134, 0.20146973407971586, -0.017117761578530566, -3.1415327532565667, 1.0693642370029629E-4]" "noBreak"
  global tool_w0_6=p[-0.6421144476781483, 0.6662879733766134, 0.20146973407971586, -0.017117761578530566, -3.1415327532565667, 1.0693642370029629E-4]
  $ 291 "tool_w5_6≔p[-0.6421260084190709, 0.66626936215097, 0.20144070436964534, 0.01707995256586941, 3.1415293685776366, -1.3993269374544494E-4]" "noBreak"
  global tool_w5_6=p[-0.6421260084190709, 0.66626936215097, 0.20144070436964534, 0.01707995256586941, 3.1415293685776366, -1.3993269374544494E-4]
  $ 292 "Moving to Waypoints" "noBreak"
  $ 293 "'Setting Change TCP'" "noBreak"
  # 'Setting Change TCP'
  $ 294 "set_change_tc_6≔aaa_set_change_tcp(tool_id_6)" "noBreak"
  global set_change_tc_6= aaa_set_change_tcp (tool_id_6)
  $ 295 "set_user_pc_6≔aaa_set_user_payload(tool_id_6)" "noBreak"
  global set_user_pc_6= aaa_set_user_payload (tool_id_6)
  $ 296 "'Exit Path'" "noBreak"
  # 'Exit Path'
  $ 297 "MoveL" "noBreak"
  $ 298 "tool_w5_6" "noBreak"
  movel(tool_w5_6, a=1.2, v=0.25)
  $ 299 "MoveL" "noBreak"
  $ 300 "tool_w4_6" "noBreak"
  movel(tool_w4_6, a=1.2, v=0.25, r=0.005)
  $ 301 "AAA script at W4" "noBreak"
  $ 302 "set_tool_volt_6≔set_tool_voltage(0)" "noBreak"
  global set_tool_volt_6= set_tool_voltage (0)
  $ 303 "MoveL" "noBreak"
  $ 304 "tool_w3_6" "noBreak"
  movel(tool_w3_6, a=0.2, v=0.02, r=0.01)
  $ 305 "Set Change Payload and COG" "noBreak"
  $ 306 "set_change_pc_6≔aaa_set_change_payload(tool_id_6)" "noBreak"
  global set_change_pc_6= aaa_set_change_payload (tool_id_6)
  $ 307 "tool_w2_6" "noBreak"
  movel(tool_w2_6, a=0.2, v=0.02)
  $ 308 "AAA script at W1" "noBreak"
  $ 309 "'Setting voltage to 0'" "noBreak"
  # 'Setting voltage to 0'
  $ 310 "set_w1_volt_6≔set_tool_voltage(0)" "noBreak"
  global set_w1_volt_6= set_tool_voltage (0)
  $ 311 "tool_w1_6" "noBreak"
  movel(tool_w1_6, a=0.2, v=0.02)
  $ 312 "'Enter Path'" "noBreak"
  # 'Enter Path'
  $ 313 "MoveL" "noBreak"
  $ 314 "tool_w0_6" "noBreak"
  movel(tool_w0_6, a=1.2, v=0.25)
  # end: URCap Program Node
end
